// TIA Portal V16 export
// export: Created 2025-12-18T09:31:57.6763017Z, ExportSetting WithDefaults, DisplayName Totally Integrated Automation Portal, DisplayVersion V16, DisplayName TIA Portal Version Control Interface, DisplayVersion V16, DisplayName TIA Portal Openness, DisplayVersion V16, DisplayName STEP 7 Professional, DisplayVersion V16, DisplayName STEP 7 Safety, DisplayVersion V16, DisplayName WinCC Advanced, DisplayVersion V16
TYPE "UDT SDManager"
// stored: IsFailsafeCompliant false
   STRUCT
      Status : Struct
         DownloadedData : Array[0..2] of Int;
         xTiaReady : Bool;
         xCReady : Bool;
         xDataTransfered : Bool;
      END_STRUCT;
      Command : Struct
         xSpare : Bool;
      END_STRUCT;
      Fault : Struct
         xSpare : Bool;
      END_STRUCT;
   END_STRUCT;
END_TYPE
